{attribute 'GeneratedUsingTerminal: EL6201-0000-0017'}
{attribute addProperty BoxType "EL6201-0000-0017"}
{attribute addProperty Id "Slave_14A_DI0BOOL1Slave_14A_DI1BOOL1Slave_14A_DI2BOOL1Slave_14A_DI3BOOL1Slave_14B_DI0BOOL1Slave_14B_DI1BOOL1Slave_14B_DI2BOOL1Slave_14B_DI3BOOL1"}
{attribute addProperty CRC "1122987788"}
{attribute addProperty Size "8"}
TYPE Slave_14_Inputs_42EF6F0C :
STRUCT
	{attribute addProperty Name "Slave_14A_DI0"}
	Slave_14A_DI0 : BOOL;
	{attribute addProperty Name "Slave_14A_DI1"}
	Slave_14A_DI1 : BOOL;
	{attribute addProperty Name "Slave_14A_DI2"}
	Slave_14A_DI2 : BOOL;
	{attribute addProperty Name "Slave_14A_DI3"}
	Slave_14A_DI3 : BOOL;
	{attribute addProperty Name "Slave_14B_DI0"}
	Slave_14B_DI0 : BOOL;
	{attribute addProperty Name "Slave_14B_DI1"}
	Slave_14B_DI1 : BOOL;
	{attribute addProperty Name "Slave_14B_DI2"}
	Slave_14B_DI2 : BOOL;
	{attribute addProperty Name "Slave_14B_DI3"}
	Slave_14B_DI3 : BOOL;
END_STRUCT
END_TYPE

(* stored: Version 1.2.0.0, ProductVersion 3.1.4024.9
   DUT Slave_14_Inputs_42EF6F0C: Id {ea4b71fe-5009-45b6-bf67-c370132ff83d} *)
